FUNCTION_BLOCK FB_DCSwitchgear
VAR_INPUT
END_VAR
VAR_OUTPUT
	get		: ST_DCSwitchgear_get;
END_VAR
VAR
END_VAR

END_FUNCTION_BLOCK

(* stored: Version 1.1.0.1, ProductVersion 3.1.4024.12
   POU FB_DCSwitchgear: Id {dd571d5c-e744-4b94-9f6f-9bb8e17dc6de}, SpecialFunc None *)
